(* PLC project Blank Project, Blank Blank 1.0 *)
(* stored: creationDateTime 2016-05-18T21:14:07, modificationDateTime 2018-07-31T15:32:01 *)

PROGRAM My_Program
  VAR
    high_sensor_pin AT %IX0.3 : BOOL;
    flow_pin AT %QX0.0 : BOOL;
    manual_flow AT %QX1.2 : BOOL;
    manual_pump AT %QX1.1 : BOOL;
    manual AT %QX0.7 : BOOL;
    low_sensor_pin AT %IX0.6 : BOOL;
    pump_pin AT %QX0.1 : BOOL;
  END_VAR

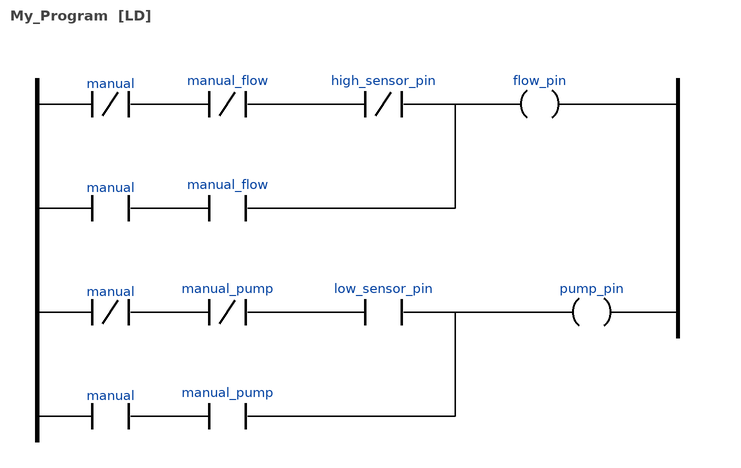
(* LD diagram, written out as Structured Text *)
flow_pin := NOT manual AND NOT manual_flow AND NOT high_sensor_pin OR manual AND manual_flow;
pump_pin := NOT manual AND NOT manual_pump AND low_sensor_pin OR manual AND manual_pump;
END_PROGRAM

CONFIGURATION Config0
  RESOURCE Res0 ON PLC
    TASK TaskMain(INTERVAL := T#5s0ms, PRIORITY := 0);
    PROGRAM Inst0 WITH TaskMain : My_Program;
  END_RESOURCE
END_CONFIGURATION
